KUKA KRL program: trabalho_concluido.src

&ACCESS RVO11
&REL 2
&PARAM TEMPLATE = C:\KRC\Roboter\Template\ExpertVorgabe
&PARAM EDITMASK = *
DEF trabalho_concluido( )


;FOLD ; FIM DO PROCESSO DE SOLDAGEM;%{PE}%R 4.1.16,%MKUKATPBASIS,%CCOMMENT,%VNORMAL,%P 2:FIM DO PROCESSO DE SOLDAGEM
;ENDFOLD
;FOLD PULSE 3333 'R1_Trabalho Concluido' State=TRUE Time=3 sec;%{PE}%R 8.2.20,%MKUKATPBASIS,%COUT,%VPULSE,%P 2:3333, 3:R1_Trabalho Concluido, 5:TRUE, 6:, 8:3
PULSE($OUT[3333], TRUE,3)
;ENDFOLD

END
